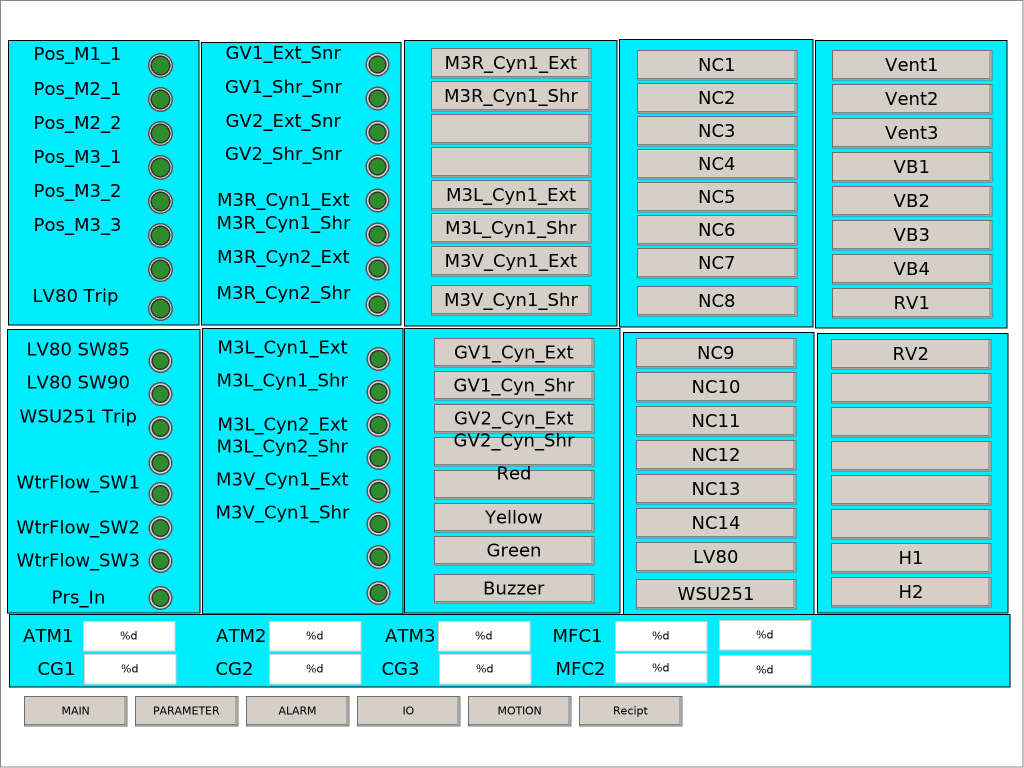
VISUALIZATION IO_TABLE  // 1024x768, background image ImagePool_Base.base
    RoundedRectangle (623,332 191x283)
    RoundedRectangle (619,39 194x288)
    RoundedRectangle (817,333 191x280)
    RoundedRectangle (8,40 191x285)
    Lamp1 (146,83 29x33), variable: DI0_1, style: Lamp-Lamp1-Green
    Lamp1 (146,117 29x33), variable: DI0_2, style: Lamp-Lamp1-Green
    Lamp1 (146,49 29x33), variable: DI0_0, style: Lamp-Lamp1-Green
    Lamp1 (146,185 29x33), variable: DI0_4, style: Lamp-Lamp1-Green
    Lamp1 (146,151 29x33), variable: DI0_3, style: Lamp-Lamp1-Green
    Lamp1 (146,292 29x33), variable: DI0_7, style: Lamp-Lamp1-Green
    Lamp1 (146,253 29x33), variable: DI0_6, style: Lamp-Lamp1-Green
    Lamp1 (146,219 29x33), variable: DI0_5, style: Lamp-Lamp1-Green
    Label (-9,50 173x30), "Pos_M1_1"
    Label (-9,85 173x30), "Pos_M2_1"
    Label (-9,119 173x30), "Pos_M2_2"
    Label (-9,153 173x30), "Pos_M3_1"
    Label (-9,187 173x30), "Pos_M3_2"
    Label (-9,221 173x30), "Pos_M3_3"
    Label (-9,255 173x30)
    Label (-11,292 173x30), "LV80 Trip"
    RoundedRectangle (7,329 193x284)
    Lamp1 (147,378 27x32), variable: DI1_1, style: Lamp-Lamp1-Green
    Lamp1 (147,412 27x32), variable: DI1_2, style: Lamp-Lamp1-Green
    Lamp1 (147,345 27x32), variable: DI1_0, style: Lamp-Lamp1-Green
    Lamp1 (147,478 27x32), variable: DI1_4, style: Lamp-Lamp1-Green
    Lamp1 (147,447 27x32), variable: DI1_3, style: Lamp-Lamp1-Green
    Lamp1 (147,582 27x32), variable: DI1_7, style: Lamp-Lamp1-Green
    Lamp1 (147,545 27x32), variable: DI1_6, style: Lamp-Lamp1-Green
    Lamp1 (147,512 27x32), variable: DI1_5, style: Lamp-Lamp1-Green
    Label (-2,346 161x29), "LV80 SW85"
    Label (-2,379 161x29), "LV80 SW90"
    Label (-2,413 161x29), "WSU251 Trip"
    Label (-2,443 161x29)
    Label (-2,479 161x29), "WtrFlow_SW1"
    Label (-2,513 161x29), "WtrFlow_SW2"
    Label (-2,546 161x29), "WtrFlow_SW3"
    Label (-2,583 161x29), "Prs_In"
    RoundedRectangle (815,40 192x288)
    RoundedRectangle (9,614 1001x73)
    RoundedRectangle (201,42 200x283)
    Lamp1 (364,82 27x33), variable: DI2_1, style: Lamp-Lamp1-Green
    Lamp1 (364,116 27x33), variable: DI2_2, style: Lamp-Lamp1-Green
    Lamp1 (364,48 27x33), variable: DI2_0, style: Lamp-Lamp1-Green
    Lamp1 (364,184 27x33), variable: DI2_4, style: Lamp-Lamp1-Green
    Lamp1 (364,150 27x33), variable: DI2_3, style: Lamp-Lamp1-Green
    Lamp1 (364,252 27x33), variable: DI2_6, style: Lamp-Lamp1-Green
    Lamp1 (364,218 27x33), variable: DI2_5, style: Lamp-Lamp1-Green
    Lamp1 (364,288 27x33), variable: DI2_7, style: Lamp-Lamp1-Green
    Label (196,49 175x30), "GV1_Ext_Snr"
    Label (196,83 175x30), "GV1_Shr_Snr"
    Label (196,117 175x30), "GV2_Ext_Snr"
    Label (196,150 175x30), "GV2_Shr_Snr"
    Label (196,185 175x30), "M3R_Cyn1_Ext"
    Label (196,219 175x30), "M3R_Cyn1_Shr"
    Label (196,253 175x30), "M3R_Cyn2_Ext"
    Label (196,289 175x30), "M3R_Cyn2_Shr"
    RoundedRectangle (202,328 201x286)
    Lamp1 (365,376 27x32), variable: DI3_1, style: Lamp-Lamp1-Green
    Lamp1 (365,409 27x32), variable: DI3_2, style: Lamp-Lamp1-Green
    Lamp1 (365,343 27x32), variable: DI3_0, style: Lamp-Lamp1-Green
    Lamp1 (365,475 27x32), variable: DI3_4, style: Lamp-Lamp1-Green
    Lamp1 (365,442 27x32), variable: DI3_3, style: Lamp-Lamp1-Green
    Lamp1 (365,541 27x32), variable: DI3_6, style: Lamp-Lamp1-Green
    Lamp1 (365,508 27x32), variable: DI3_5, style: Lamp-Lamp1-Green
    Lamp1 (365,577 27x32), variable: DI3_7, style: Lamp-Lamp1-Green
    Label (195,344 175x29), "M3L_Cyn1_Ext"
    Label (195,377 175x29), "M3L_Cyn1_Shr"
    Label (195,410 175x29), "M3L_Cyn2_Ext"
    Label (195,443 175x29), "M3L_Cyn2_Shr"
    Label (195,476 175x29), "M3V_Cyn1_Ext"
    Label (195,509 175x29), "M3V_Cyn1_Shr"
    RoundedRectangle (404,40 213x286)
    Button (431,48 160x30), "M3R_Cyn1_Ext"
        toggle DO0_0
    Button (431,81 160x30), "M3R_Cyn1_Shr"
        toggle DO0_1
    Button (431,114 160x30)
        toggle DO0_2
    Button (431,147 160x30)
        toggle DO0_3
    Button (431,180 160x30), "M3L_Cyn1_Ext"
        toggle DO0_4
    Button (431,213 160x30), "M3L_Cyn1_Shr"
        toggle DO0_5
    Button (431,246 160x30), "M3V_Cyn1_Ext"
        toggle DO0_6
    Button (431,285 160x30), "M3V_Cyn1_Shr"
        toggle DO0_7
    RoundedRectangle (404,328 216x285)
    Button (434,338 160x29), "GV1_Cyn_Ext"
        toggle DO1_0
    Button (434,371 160x29), "GV1_Cyn_Shr"
        toggle DO1_1
    Button (434,404 160x29), "GV2_Cyn_Ext"
        toggle DO1_2
    Button (434,437 160x29), "GV2_Cyn_Shr"
        toggle DO1_3
    Button (434,470 160x29), "Red"
        toggle DO1_4
    Button (434,503 160x29), "Yellow"
        toggle DO1_5
    Button (434,536 160x29), "Green"
        toggle DO1_6
    Button (434,574 160x29), "Buzzer"
        toggle DO1_7
    Button (637,50 160x30), "NC1"
        toggle DO2_0
    Button (637,83 160x30), "NC2"
        toggle DO2_1
    Button (637,116 160x30), "NC3"
        toggle DO2_2
    Button (637,149 160x30), "NC4"
        toggle DO2_3
    Button (637,182 160x30), "NC5"
        toggle DO2_4
    Button (637,215 160x30), "NC6"
        toggle DO2_5
    Button (637,248 160x30), "NC7"
        toggle DO2_6
    Button (637,286 160x30), "NC8"
        toggle DO2_7
    Button (636,338 160x30), "NC9"
        toggle DO3_0
    Button (636,372 160x30), "NC10"
        toggle DO3_1
    Button (636,406 160x30), "NC11"
        toggle DO3_2
    Button (636,440 160x30), "NC12"
        toggle DO3_3
    Button (636,474 160x30), "NC13"
        toggle DO3_4
    Button (636,508 160x30), "NC14"
        toggle DO3_5
    Button (636,542 160x30), "LV80"
        toggle DO3_6
    Button (636,579 160x30), "WSU251"
        toggle DO3_7
    Button (832,50 160x30), "Vent1"
        toggle DO4_0
    Button (832,84 160x30), "Vent2"
        toggle DO4_1
    Button (832,118 160x30), "Vent3"
        toggle DO4_2
    Button (832,152 160x30), "VB1"
        toggle DO4_3
    Button (832,186 160x30), "VB2"
        toggle DO4_4
    Button (832,220 160x30), "VB3"
        toggle DO4_5
    Button (832,254 160x30), "VB4"
        toggle DO4_6
    Button (832,288 160x30), "RV1"
        toggle DO4_7
    Button (831,339 160x30), "RV2"
        toggle DO5_0
    Button (831,373 160x30)
        toggle DO5_1
    Button (831,407 160x30)
        toggle DO5_2
    Button (831,441 160x30)
        toggle DO5_3
    Button (831,475 160x30)
        toggle DO5_4
    Button (831,509 160x30)
        toggle DO5_5
    Button (831,543 160x30), "H1"
        toggle DO5_6
    Button (831,577 160x30), "H2"
        toggle DO5_7
    Label (821,398 161x30)
    Label (821,432 161x30)
    Label (821,466 161x30)
    Label (821,500 161x30)
    Label (821,534 161x30)
    Textfield (83,621 92x30), "%d", text variable: AI0_0
        OnMouseClick: write the text variable via Default, min 0, max 300
    Textfield (269,621 92x30), "%d", text variable: AI0_1
        OnMouseClick: write the text variable via Default, min 0, max 300
    Textfield (438,621 92x30), "%d", text variable: AI0_2
        OnMouseClick: write the text variable via Default, min 0, max 300
    Textfield (84,654 92x30), "%d", text variable: AI0_3
        OnMouseClick: write the text variable via Default, min 0, max 300
    Textfield (269,654 92x30), "%d", text variable: AI1_0
        OnMouseClick: write the text variable via Default, min 0, max 300
    Textfield (439,654 92x30), "%d", text variable: AI1_1
        OnMouseClick: write the text variable via Default, min 0, max 300
    Textfield (615,621 92x30), "%d", text variable: AI1_2
    Textfield (615,653 92x30), "%d", text variable: AI1_3
    Label (21,621 55x30), "ATM1"
    Label (214,621 55x30), "ATM2"
    Label (383,621 55x30), "ATM3"
    Label (29,654 55x30), "CG1"
    Label (207,654 55x30), "CG2"
    Label (373,654 55x30), "CG3"
    Label (550,621 55x30), "MFC1"
    Label (553,654 55x30), "MFC2"
    Textfield (719,620 92x30), "%d", text variable: AO0_2
        OnMouseClick: write the text variable via Default, min 0, max 300
    Textfield (719,655 92x30), "%d", text variable: AO0_3
        OnMouseClick: write the text variable via Default, min 0, max 300
    Button (24,696 103x30), "MAIN"
        OnMouseClick: change screen: MainBase
    Button (135,696 103x30), "PARAMETER"
        OnMouseClick: change screen: PARAMETER
    Button (246,696 103x30), "ALARM"
        OnMouseClick: change screen: ALARM
    Button (357,696 103x30), "IO"
        OnMouseClick: change screen: IO_TABLE
    Button (468,696 103x30), "MOTION"
        OnMouseClick: change screen: MOTION
    Button (579,696 103x30), "Recipt"
        OnMouseClick: change screen: Recipt
END_VISUALIZATION

(* stored: Version 1.1.0.1, ProductVersion 3.1.4024.11
   Visu IO_TABLE: Id {debefc24-95d0-4525-b4fa-d6c8d2f2d93f} *)
